FUNCTION_BLOCK Interlock
VAR
	_Locked : BOOL;
END_VAR

METHOD Lock : BOOL
VAR_INPUT
END_VAR
_Locked := TRUE;
END_METHOD

PROPERTY Locked : bool
GET
Locked := _Locked;
END_GET
END_PROPERTY

METHOD Unlock : BOOL
VAR_INPUT
END_VAR
_Locked := false;
END_METHOD

PROPERTY Unlocked : bool
GET
Unlocked := NOT _Locked;
END_GET
END_PROPERTY

END_FUNCTION_BLOCK

(* stored: Version 1.1.0.1, ProductVersion 3.1.4024.12
   POU Interlock: Id {2fdb8b3a-37c3-426f-9e81-673159b1ccfe}, SpecialFunc None
   Method Lock: Id {4ddb4347-23aa-417a-a71b-3dc70fac702e}
   Property Locked: Id {6425f6cf-50a4-4dfb-a771-1d6e114ee8fa}
   Get Get: Id {87fa3bfd-2342-4971-afd5-ff18b0c2e640}
   Method Unlock: Id {6580c073-0cb3-4d75-876d-930fa523d908}
   Property Unlocked: Id {50b4c469-df3e-4820-94b4-f49b904bc837}
   Get Get: Id {8faa066b-b816-480c-851e-1d3de346bbee} *)
